// TIA Portal V17 export
// export: Created 2025-03-07T09:24:04.6569162Z, ExportSetting WithDefaults, DisplayName Totally Integrated Automation Portal, DisplayVersion V17 Update 8, DisplayName TIA Portal Openness, DisplayVersion V17 Update 8, DisplayName TIA Portal Version Control Interface, DisplayVersion V17, DisplayName SINAMICS Startdrive Advanced, DisplayVersion V17 SP2, DisplayName SINAMICS Startdrive G110M, G120, G120C, G120D, G120P, G115D, DisplayVersion V17 SP2, DisplayName SINAMICS Startdrive G130, G150, S120, S150, SINAMICS MV, S210, DisplayVersion V17 SP2, DisplayName STEP 7 Professional, DisplayVersion V17 Update 8, DisplayName SINUMERIK ONE STEP 7 Toolbox, DisplayVersion V17 Update 12, DisplayName SINUMERIK 840D sl STEP 7 Toolbox, DisplayVersion V17 Update 12, DisplayName STEP 7 Safety, DisplayVersion V17 Update 6, DisplayName WinCC Advanced, DisplayVersion V17 Update 8
DATA_BLOCK "DB21205_UNIT_01_COMBINER_MEDICOAT"   // DB21205
{ DB_Accessible_From_OPC_UA := 'FALSE' }
VERSION : 0.1
// stored: AutoNumber false, DBAccessibleFromOPCUA false, DBAccessibleFromWebserver true, InstanceOfName FB21200_POWDER_FLOW_SENSOR_MEDICOAT, InstanceOfType FB
"FB21200_POWDER_FLOW_SENSOR_MEDICOAT"
   // VAR_INPUT
   //    ANALOG_VALUE : Int := 5;
   //    TIMER_1 : Timer := T33;
   //    POWDER_FEEDER_ON { ExternalVisible := 'False'; ExternalWritable := 'False'} : Bool := FALSE;
   // END_VAR
   // VAR_OUTPUT
   //    POWDER_FLOW_ON : Bool := TRUE;
   //    NO_POWDER_FLOW_ALARM : Bool := FALSE;
   //    WARNING_LIMIT : Bool := FALSE;
   //    ERROR_CONFIGURATION : Bool := FALSE;
   // END_VAR
   // VAR RETAIN
   //    OUTPUT : Struct
   //       VALUE_REAL : Real := 0.01525925;
   //       VALUE_INT : Int;
   //    END_STRUCT;
   //    INPUT_SETTINGS : Struct
   //       LOW_RANGE : Real := 0.0;
   //       HIGH_RANGE : Real := 10.0;
   //       LOW_LIMIT_TO_POWDER_FLOW_ON : Real := 0.0;
   //       UNIT_NUMBER : Int;
   //       FEEDER_NUMBER : Int;
   //    END_STRUCT;
   //    ALARMS_SETTINGS : Struct
   //       WARN_LIMIT_LOW : Real := 0.0;
   //       WARN_LIMIT_HIGH : Real := 100.0;
   //    END_STRUCT;
   //    LOG : Struct
   //       DATE_MAX_MASS : Date_And_Time := DT#1990-01-01-00:00:00;
   //       VALUE_MAX_MASS : Real := 0.0;
   //    END_STRUCT;
   // END_VAR
BEGIN
END_DATA_BLOCK
